TYPE u_SM6020 :
UNION
	total: ARRAY[0..3] OF BYTE;
	rtotal			:REAL;// totalizado

END_UNION
END_TYPE

(* stored: Version 1.1.0.1, ProductVersion 3.1.4024.12
   DUT u_SM6020: Id {4d8ba378-aba8-42c2-bc16-33a9a26fbfda} *)
